// TIA Portal V19 export
FUNCTION "TEST FILLING PRESSUR." : Void   // FC17, STL
TITLE = TEST FILLING PRESSURE
{ S7_Optimized_Access := 'TRUE' }
NAME : TSTFILLI
VERSION : 0.0
// Comment
// stored: AutoNumber false
BEGIN

NETWORK
TITLE = TEST FILLING PRESSURE
      A     "TEST FILLING PRESSURE";
      JC    M001;
      R     "DUMMY TEST PT 01.67";
      BEU;
M001: AN    "S0 PRESTERILIZING";
      JC    END;
      AN    "AutoPT0167/IP0149";
      BEC;
      L     "MeasuredValues".PT0167REAL;  //"DB-ANALOG INPUT".PT0167MeasPressure
      L     "Setpoints".MinPresUnsterile;  //"DB SETPOINTS".MinPresUnsterile
      >R;
      BEC;
      R     "S7 PRESTERILIZING";
      R     "S6 PRESTERILIZING";
      R     "S5 PRESTERILIZING";
      R     "S4 PRESTERILIZING";
      R     "S3 PRESTERILIZING";
      R     "S2 PRESTERILIZING";
      R     "S1 PRESTERILIZING";
      R     "TEST FILLING PRESSURE";
      S     "ProcessAndPbAlarms"."A"[44];  //A44_FillPressureTooLow// filling pressure too low
      BEU;
END:  NOP   0;

NETWORK
TITLE = DUMMY TEST FILLING PRESSURE
      A     "S0 PRODUCTION TANK";
      JC    M000;
      R     "DUMMY TEST PT 01.67";
      BEU;
M000: AN    "TANK STERILE";
      BEC;
      L     "MeasuredValues".PT0167REAL;  // "DB-ANALOG INPUT".PT0167MeasPressure
      L     "Setpoints".MinPresUnsterile;  //"DB SETPOINTS".MinPresUnsterile
      >R;
      JC    c001;
      AN    "DUMMY TEST PT 01.67";
      S     "DUMMY TEST PT 01.67";
      S     "TIM35";
      BEC;
      A     "T 35 DELAY PT 01.67";
      BEC;
      S     "ProcessAndPbAlarms"."A"[44];  //A44_FillPressureTooLow// filling press too low
      R     "TANK STERILE";
      R     "TEST FILLING PRESSURE";
      BEU;
c001: R     "DUMMY TEST PT 01.67";
      L     "MeasuredValues".PT0167REAL;  // "DB-ANALOG INPUT".PT0167MeasPressure
      L     "Setpoints".PT0167LowPressure;  //"DB SETPOINTS".PT0167LowPressure
      >R;
      BEC;
      S     "ProcessAndPbAlarms"."A"[45];  //A45_FillingPressureLow
      BEU;
END_FUNCTION
